Yaskawa INFORM job: WIRE-CUTTER-LONG-45.JBI

/JOB
//NAME WIRE-CUTTER-LONG-45
///FOLDERNAME CLEAN
//POS
///NPOS 7,0,0,0,0,0
///TOOL 4
///POSTYPE PULSE
///PULSE
C00000=76555,-57488,-86646,-37317,-91588,59090
C00001=91260,-41973,-78038,-42101,-83430,56373
C00002=89708,-30876,-81531,-42313,-78166,59136
C00003=88706,-36118,-84980,-41893,-78994,59170
C00004=87986,-39534,-87102,-41591,-79618,59187
C00005=88167,-48754,-78974,-41066,-86966,56210
C00006=67013,-73974,-65084,-37660,-113120,55534
//INST
///DATE 2021/10/29 11:50
///ATTR SC,RO
///GROUP1 RB1
NOP
MOVJ C00000 VJ=75.00
MOVJ C00001 VJ=25.00
'WIRE CUTER
'CUT WIRE AT 15mm
PULSE OT#(4095) T=3.00
TIMER T=3.00
MOVJ C00002 VJ=15.00
MOVL C00003 V=21.2 PL=0
TIMER T=0.50
MOVL C00004 V=42.3 PL=0
TIMER T=0.50
MOVL C00005 V=211.7
MOVJ C00006 VJ=75.00
END
